FUNCTION_BLOCK _FLOAT_TestSuite EXTENDS TcUnit.FB_TestSuite
VAR
END_VAR

TestAddress();
TestClearReference();
TestClone();
TestIdentifierReturnsExpected();
TestIecTypeReturnsExpected();
TestMakeReferenceToFollowsReference();
TestMakeReferenceToUpdatesReference();
TestSize();
TestValueReturnsExpectedAfterInit();
TestValueReturnsExpectedAfterChange();
TestSerializeTypeWith();
TestSerializeWith();
TestTryDeserializeFrom();
TestTryMakeReferenceToFollowsReference();
TestTryMakeReferenceToUpdatesReference();

METHOD PUBLIC TestAddress
VAR
    _type : _FLOAT(0);
    notExpected : PVOID := 0;
    actual : PVOID;
END_VAR
TEST('TestAddress');

actual := _type.Address;

AssertFalse(
    Condition := (notExpected = actual),
    Message := 'Type did not return a valid address.'
);

TEST_FINISHED();
END_METHOD

METHOD PUBLIC TestClearReference
VAR
    _type : _FLOAT(S_OK);
	target : FLOAT := 0;
    expected : FLOAT := 0;
    actual : FLOAT;
END_VAR
TEST('TestClearReference');

_type.MakeReferenceTo(target);
_type.ClearReference();
target := 123.4;

actual := _type.Value;

AssertEquals_LREAL(
    Expected := expected,
    Actual := actual,
    Delta := LREAL#0.001,
    Message := 'Value did not follow target change'
);

TEST_FINISHED();
END_METHOD

METHOD PUBLIC TestClone
VAR
    _type : _FLOAT(0);
	clone : I_Datatype;
	isValidClone : BOOL;
	compareResult : DINT;
END_VAR
TEST('TestClone');

clone := _type.Clone();

isValidClone := clone <> 0;

IF isValidClone THEN
	compareResult := memcmp(_type.Address, clone.Address, clone.Size);
END_IF

AssertTrue(
	Condition := isValidClone,
	Message := 'Clone did not produce a clone'
);

AssertEquals_DINT(
	Expected := 0,
    Actual := compareResult,
    Message := 'Clone did not return a valid clone.'
);

clone.Dispose();

TEST_FINISHED();
END_METHOD

METHOD PUBLIC TestIdentifierReturnsExpected
VAR
    _type : _FLOAT(0);
    expected : STRING := 'FLOAT';
    actual : STRING;
END_VAR
TEST('TestIdentifierReturnsExpected');

actual := _type.Identifier;

AssertEquals_STRING(
    Expected := expected,
    Actual := actual,
    Message := 'Type did not return correct iec type.'
);

TEST_FINISHED();
END_METHOD

METHOD PUBLIC TestIecTypeReturnsExpected
VAR
    _type : _FLOAT(0);
    expected : STRING := 'ALIAS';
    actual : STRING;
END_VAR
TEST('TestIecTypeReturnsExpected');

actual := _type.IecType;

AssertEquals_STRING(
    Expected := expected,
    Actual := actual,
    Message := 'Type did not return correct iec type.'
);

TEST_FINISHED();
END_METHOD

METHOD PUBLIC TestMakeReferenceToFollowsReference
VAR
    _type : _FLOAT(0);
	target : FLOAT := 0;
    expected : FLOAT := 123.4;
    actual : FLOAT;
END_VAR
TEST('TestMakeReferenceToFollowsReference');

_type.MakeReferenceTo(target);
target := 123.4;

actual := _type.Value;

AssertEquals_LREAL(
    Expected := expected,
    Actual := actual,
    Delta := LREAL#0.001,
    Message := 'Value did not follow target change'
);

TEST_FINISHED();
END_METHOD

METHOD PUBLIC TestMakeReferenceToUpdatesReference
VAR
    _type : _FLOAT(0);
	target : FLOAT := 0;
    expected : FLOAT := 123.4;
    actual : FLOAT;
END_VAR
TEST('TestMakeReferenceToUpdatesReference');

_type.MakeReferenceTo(target);
_type.Value := 123.4;

actual := target;

AssertEquals_LREAL(
    Expected := expected,
    Actual := actual,
    Delta := LREAL#0.001,
    Message := 'Value did not update target'
);

TEST_FINISHED();
END_METHOD

METHOD PUBLIC TestSerializeTypeWith
VAR
    _type : _FLOAT(0);
    serializer : JsonSerializer;
    expected : STRING := '{"name":"FLOAT","type":"ALIAS","baseType":{"type":"LREAL"}}';
    actual : STRING(500);
END_VAR
TEST('TestSerializeTypeWith');

serializer.Reset();
_type.SerializeTypeWith(serializer);
serializer.TryGetSerializedData(ADR(actual), SIZEOF(actual));

AssertEquals_STRING(
    Expected := expected,
    Actual := actual,
    Message := 'Serialization of type did not return correct string.'
);

TEST_FINISHED();
END_METHOD

METHOD PUBLIC TestSerializeWith
VAR
    _type : _FLOAT(123.4);
    serializer : JsonSerializer;
    expected : STRING := '123.4';
    actual : STRING(500);
END_VAR
TEST('TestSerializeWith');

serializer.Reset();
_type.SerializeWith(serializer);
serializer.TryGetSerializedData(ADR(actual), SIZEOF(actual));

AssertEquals_STRING(
    Expected := expected,
    Actual := actual,
    Message := 'Serialization of type data did not return correct string.'
);

TEST_FINISHED();
END_METHOD

METHOD PUBLIC TestSize
VAR
    _type : _FLOAT(0);
    expected : UDINT := SIZEOF(FLOAT);
    actual : UDINT;
END_VAR
TEST('TestSize');

actual := _type.Size;

AssertEquals_UDINT(
    Expected := Expected,
    Actual := actual,
    Message := 'Type did not return the correct size.'
);

TEST_FINISHED();
END_METHOD

METHOD PUBLIC TestTryDeserializeFrom
VAR
    deserializer : JsonDeserializer;
    feedback : DeserializerFeedback;
    json : STRING := '123.4';
    _type : _FLOAT(0.0);
    expected : FLOAT := 123.4;
    actual : FLOAT;
 END_VAR
TEST('TestTryDeserializeFrom');

deserializer.Reset();
deserializer.TryLoad(json);
_type.TryDeserializeFrom(Deserializer, Feedback);

actual := _type.Value;

AssertEquals_LREAL(
    Expected := expected,
    Actual := actual,
    Delta := LREAL#0.001,
    Message := 'Type did not deserialize correctly.'
);

TEST_FINISHED();
END_METHOD

METHOD PUBLIC TestTryMakeReferenceToFollowsReference
VAR
    _type : _FLOAT(0.0);
	target : _FLOAT(0.0);
    expected : FLOAT := 123.4;
    actual : FLOAT;
END_VAR
TEST('TestTryMakeReferenceToFollowsReference');

_type.TryMakeReferenceTo(target);
target.Value := 123.4;

actual := _type.Value;

AssertEquals_LREAL(
    Expected := expected,
    Actual := actual,
    Delta := LREAL#0.001,
    Message := 'Value did not follow target change'
);

TEST_FINISHED();
END_METHOD

METHOD PUBLIC TestTryMakeReferenceToUpdatesReference
VAR
    _type : _FLOAT(0.0);
	target : _FLOAT(0.0);
    expected : FLOAT := 123.4;
    actual : FLOAT;
END_VAR
TEST('TestTryMakeReferenceToUpdatesReference');

_type.TryMakeReferenceTo(target);
_type.Value := 123.4;

actual := target.Value;

AssertEquals_LREAL(
    Expected := expected,
    Actual := actual,
    Delta := LREAL#0.001,
    Message := 'Value did not update target'
);

TEST_FINISHED();
END_METHOD

METHOD PUBLIC TestValueReturnsExpectedAfterChange
VAR
    _type : _FLOAT(0.0);
    expected : FLOAT := 123.4;
    actual : FLOAT;
END_VAR
TEST('TestValueReturnsExpectedAfterChange');

_type.Value := 123.4;

actual := _type.Value;

AssertEquals_LREAL(
    Expected := expected,
    Actual := actual,
    Delta := LREAL#0.001,
    Message := 'Expected value not returned after change.'
);

TEST_FINISHED();
END_METHOD

METHOD PUBLIC TestValueReturnsExpectedAfterInit
VAR
    _type : _FLOAT(123.4);
    expected : FLOAT := 123.4;
    actual : FLOAT;
END_VAR
TEST('TestValueReturnsExpectedAfterInit');

actual := _type.Value;

AssertEquals_LREAL(
    Expected := expected,
    Actual := actual,
    Delta := LREAL#0.001,
    Message := 'Expected value not returned after Init.'
);

TEST_FINISHED();
END_METHOD

END_FUNCTION_BLOCK

(* stored: Version 1.1.0.1, ProductVersion 3.1.4024.12
   POU _FLOAT_TestSuite: Id {79c7deeb-7586-0780-1c9d-9f7986e3a47f}, SpecialFunc None
   Method TestAddress: Id {c1d840d9-0ed6-0288-29b3-0c640a6bf4e0}
   Method TestClearReference: Id {2b3b5110-93bd-0786-2782-7d85d4c526a9}
   Method TestClone: Id {f6da8deb-7612-0dd1-1223-dea8c8b201a0}
   Method TestIdentifierReturnsExpected: Id {1317e8f6-40b2-0427-0bf6-5681b2a562b6}
   Method TestIecTypeReturnsExpected: Id {70102dc6-4c9b-01aa-0d66-858ac2276aa5}
   Method TestMakeReferenceToFollowsReference: Id {904d2976-f6aa-0838-2252-20a1ae2f02f3}
   Method TestMakeReferenceToUpdatesReference: Id {9e032db6-b5b4-064b-27d7-f7da7a9ad60d}
   Method TestSerializeTypeWith: Id {87036562-7e1f-048f-3303-f3cdfab0f065}
   Method TestSerializeWith: Id {e743a10a-4ed3-0dc0-1211-b839e9555568}
   Method TestSize: Id {05188172-760d-08a1-16ca-e12a15711f8d}
   Method TestTryDeserializeFrom: Id {485aec3e-bdae-0365-1d43-9d1f481c3a36}
   Method TestTryMakeReferenceToFollowsReference: Id {fc197e03-825f-0dc3-00b1-1688dadf72c7}
   Method TestTryMakeReferenceToUpdatesReference: Id {f3422f7c-01fb-020a-2719-c248e21fa4c0}
   Method TestValueReturnsExpectedAfterChange: Id {f3397b61-fd74-0826-3590-ff518ddaaca5}
   Method TestValueReturnsExpectedAfterInit: Id {398ae652-078b-07c8-2834-732ea2920a17} *)
